INTERFACE I_DatatypeOperation EXTENDS I_Disposable

METHOD Execute
VAR
END_VAR
END_METHOD

END_INTERFACE

(* stored: Version 1.1.0.1, ProductVersion 3.1.4024.12
   Itf I_DatatypeOperation: Id {4d749c49-3db4-4fa2-97e5-003f1b6ebe8c}
   Method Execute: Id {8c79392f-5f6c-4d1e-aa80-a516a128b16f} *)
